(* CoDeSys 2.3 export: ST_MAST_SETUP.EXP *)

(* Data type *)
TYPE ST_MAST_SETUP :
STRUCT
	Cycle : REAL; (*Seconds*)

	aFSY  : ARRAY[1..4,1..6] OF REAL;
	aBDef : ARRAY[1..4,1..6] OF REAL;
	aTDef : ARRAY[1..4,1..6] OF REAL;


END_STRUCT
END_TYPE
